// TIA Portal V15.1 export
// export: Created 2024-05-17T05:38:37.8668789Z, ExportSetting WithDefaults, DisplayName Totally Integrated Automation Portal, DisplayVersion V15.1 Update 5, DisplayName TIA Portal Openness, DisplayVersion V15.1 Update 5, DisplayName SINAMICS Startdrive Advanced, DisplayVersion V15.1, DisplayName G130, G150, S120, S150, SINAMICS MV, S210, DisplayVersion V15.1, DisplayName G110M, G120, G120C, G120D, G120P, DisplayVersion V15.1, DisplayName STEP 7 Professional, DisplayVersion V15.1 Update 5, DisplayName STEP 7 Safety, DisplayVersion V15.1, DisplayName WinCC Professional, DisplayVersion V15.1 Update 5, DisplayName SIMATIC Visualization Architect, DisplayVersion V15.1
FUNCTION_BLOCK "LGBMotor2W2S-FC302PN"   // FB6601, FBD
TITLE = LGBMotor2W2S-FC302PN
{ S7_Optimized_Access := 'TRUE' }
AUTHOR : VCC
FAMILY : Actuator
NAME : Danfoss
VERSION : 0.1
// ============================================================================
// This "LMotor2W2S-FC302PN" module is used in applications when a motor 2 way - variable 
// speed equipped with Danfoss FC302 is needed.
// The module contains: a motor loop equipped with 
// "1 Danfoss frequency converter.
// "1 safety switch.
// ============================================================================
// stored: AutoNumber false, IsIECCheckEnabled false, IsRetainMemResEnabled false, MemoryReserve 100, SetENOAutomatically False, UDAEnableTagReadback false
   VAR_INPUT
      I_EnableAlarm { ExternalAccessible := 'False'; ExternalVisible := 'False'; ExternalWritable := 'False'} : Bool;   // Enable alarm
      I_EnablePNReset { ExternalAccessible := 'False'; ExternalVisible := 'False'; ExternalWritable := 'False'} : Bool;   // Enable frequency convertor reset with
      I_AlarmResetPB { ExternalAccessible := 'False'; ExternalVisible := 'False'; ExternalWritable := 'False'} : Bool;   // Alarm reset pushbutton is activated
      I_MotorProtection { ExternalAccessible := 'False'; ExternalVisible := 'False'; ExternalWritable := 'False'} : Bool;   // Motor protection
      I_BrakeProtection { ExternalAccessible := 'False'; ExternalVisible := 'False'; ExternalWritable := 'False'} : Bool;   // Brake protection
      I_SafetySwitch { ExternalAccessible := 'False'; ExternalVisible := 'False'; ExternalWritable := 'False'} : Bool;   // Safety Switch
      I_SafetyOk { ExternalAccessible := 'False'; ExternalVisible := 'False'; ExternalWritable := 'False'} : Bool;   // Safety Ok
      I_MotionStopOk { ExternalAccessible := 'False'; ExternalVisible := 'False'; ExternalWritable := 'False'} : Bool;   // Safety Ok / The motion stop is Ok
      I_Release { ExternalAccessible := 'False'; ExternalVisible := 'False'; ExternalWritable := 'False'} : Bool := TRUE;   // Hold Motor Command
      I_LSpdSetMotorCmd { ExternalAccessible := 'False'; ExternalVisible := 'False'; ExternalWritable := 'False'} : Bool;   // Low speed Set Command from function after interlock
      I_HSpdSetMotorCmd { ExternalAccessible := 'False'; ExternalVisible := 'False'; ExternalWritable := 'False'} : Bool;   // High Speed Set Command from function after Interlock
      I_LSpdResMotorCmd { ExternalAccessible := 'False'; ExternalVisible := 'False'; ExternalWritable := 'False'} : Bool;   // Low speed Reset Command from function after interlock
      I_HSpdResMotorCmd { ExternalAccessible := 'False'; ExternalVisible := 'False'; ExternalWritable := 'False'} : Bool;   // High speed Reset Command from function after Interlock
      I_QuickStop { ExternalAccessible := 'False'; ExternalVisible := 'False'; ExternalWritable := 'False'} : Bool;   // QuickStop function; When FALSE the QuickStop of the Danfoss FC302 is Active
      I_ReleaseBrake { ExternalAccessible := 'False'; ExternalVisible := 'False'; ExternalWritable := 'False'} : Bool;   // Release brake
      I_InitDirection { ExternalAccessible := 'False'; ExternalVisible := 'False'; ExternalWritable := 'False'} : Bool;   // Initialisation of the direction
      I_SetupSelLsb { ExternalAccessible := 'False'; ExternalVisible := 'False'; ExternalWritable := 'False'} : Bool;   // Enable setpoint
      I_SetupSelMsb { ExternalAccessible := 'False'; ExternalVisible := 'False'; ExternalWritable := 'False'} : Bool;   // Enable setpoint
      I_LowSpeed { ExternalAccessible := 'False'; ExternalVisible := 'False'; ExternalWritable := 'False'} : Real;   // Low speed value (set-up %) Reference value for speed, stored in P2000 ot the SINAMICS G120
      I_HighSpeed { ExternalAccessible := 'False'; ExternalVisible := 'False'; ExternalWritable := 'False'} : Real;   // High speed value (set-up %) Reference value for speed, stored in P2000 ot the SINAMICS G120
   END_VAR
   VAR_OUTPUT
      O_BusFault { ExternalAccessible := 'False'; ExternalVisible := 'False'; ExternalWritable := 'False'} : Bool;   // Alarm
      O_MotorProtectionAlarm { ExternalAccessible := 'False'; ExternalVisible := 'False'; ExternalWritable := 'False'} : Bool;   // Motor protection Alarm
      O_BrakeProtectionAlarm { ExternalAccessible := 'False'; ExternalVisible := 'False'; ExternalWritable := 'False'} : Bool;   // Brake protection alarm
      O_SafetySwitchAlarm { ExternalAccessible := 'False'; ExternalVisible := 'False'; ExternalWritable := 'False'} : Bool;   // Safety Switch Alarm
      O_MotionStopWarning { ExternalAccessible := 'False'; ExternalVisible := 'False'; ExternalWritable := 'False'} : Bool;   // Drive fault / Motion Stop warning
      O_Alarm { ExternalAccessible := 'False'; ExternalVisible := 'False'; ExternalWritable := 'False'} : Bool;   // Alarm
      O_Warning { ExternalAccessible := 'False'; ExternalVisible := 'False'; ExternalWritable := 'False'} : Bool;   // Warning
      O_AlarmABCondition { ExternalAccessible := 'False'; ExternalVisible := 'False'; ExternalWritable := 'False'} : Bool;   // Alarm AB condition
      O_Active { ExternalAccessible := 'False'; ExternalVisible := 'False'; ExternalWritable := 'False'} : Bool;   // Motor loop Active
      O_BrakeFunction { ExternalAccessible := 'False'; ExternalVisible := 'False'; ExternalWritable := 'False'} : Bool;   // Brake Function
      O_ReadyForOperation { ExternalAccessible := 'False'; ExternalVisible := 'False'; ExternalWritable := 'False'} : Bool;   // Ready for operation
      O_ActualSpeed { ExternalAccessible := 'False'; ExternalVisible := 'False'; ExternalWritable := 'False'} : Real;   // Actual Speed
   END_VAR
   VAR_IN_OUT
      IO_Modes : "Modes";   // Modes
      H_HMI : "H_HMI";
      "H_GBMotor2W2S-FC302PN" : "H_GBMotor2W2S-FC302PN";
      C_HWSubInput { ExternalAccessible := 'False'; ExternalVisible := 'False'; ExternalWritable := 'False'} : HW_SUBMODULE;   // I/O
      C_HWSubOutput { ExternalAccessible := 'False'; ExternalVisible := 'False'; ExternalWritable := 'False'} : HW_SUBMODULE;   // I/O
      C_EnableCheckSpeed { ExternalAccessible := 'False'; ExternalVisible := 'False'; ExternalWritable := 'False'} : Bool;   // Enable check speed is OK
      C_TimeCheckSpeedOK { ExternalAccessible := 'False'; ExternalVisible := 'False'; ExternalWritable := 'False'} : DInt := 2000;   // Time check speed OK
      C_ReleaseBrakeUsed { ExternalAccessible := 'False'; ExternalVisible := 'False'; ExternalWritable := 'False'} : Bool;   // Release brake used
      C_MotorProtectionUsed { ExternalAccessible := 'False'; ExternalVisible := 'False'; ExternalWritable := 'False'} : Bool;   // Motor Protection used
      C_MotorProtectionNc { ExternalAccessible := 'False'; ExternalVisible := 'False'; ExternalWritable := 'False'} : Bool;   // Motor Protection Normally closed
      C_BrakeProtectionUsed { ExternalAccessible := 'False'; ExternalVisible := 'False'; ExternalWritable := 'False'} : Bool;   // Brake Protection used / Motor Protection used
      C_BrakeProtectionNc { ExternalAccessible := 'False'; ExternalVisible := 'False'; ExternalWritable := 'False'} : Bool;   // Motor Protection Normally closed / Brake Protection Normally closed
      C_SafetySwitchUsed { ExternalAccessible := 'False'; ExternalVisible := 'False'; ExternalWritable := 'False'} : Bool;   // Safety switch used
      C_SafetySwitchNc { ExternalAccessible := 'False'; ExternalVisible := 'False'; ExternalWritable := 'False'} : Bool;   // Safety switch Normally closed
      C_MotionStopUsed { ExternalAccessible := 'False'; ExternalVisible := 'False'; ExternalWritable := 'False'} : Bool;   // Motion Stop used
   END_VAR
   VAR
      Start { ExternalAccessible := 'False'; ExternalVisible := 'False'; ExternalWritable := 'False'} : Bool;   // Start
      Reverse { ExternalAccessible := 'False'; ExternalVisible := 'False'; ExternalWritable := 'False'} : Bool;   // Reverse
      MotorProtectionAlarm { ExternalAccessible := 'False'; ExternalVisible := 'False'; ExternalWritable := 'False'} : Bool;   // Motor protection Alarm
      BrakeProtectionAlarm { ExternalAccessible := 'False'; ExternalVisible := 'False'; ExternalWritable := 'False'} : Bool;   // Brake protection alarm
      CheckSpeedOK { ExternalAccessible := 'False'; ExternalVisible := 'False'; ExternalWritable := 'False'} : Bool;   // After this time the speed has to be reached
      SafetySwitchAlarm { ExternalAccessible := 'False'; ExternalVisible := 'False'; ExternalWritable := 'False'} : Bool;   // Safety Switch Alarm
      MotorProtectionAlarmABCond { ExternalAccessible := 'False'; ExternalVisible := 'False'; ExternalWritable := 'False'} : Bool;   // Motor protection Alarm condition
      BrakeProtectionAlarmABCond { ExternalAccessible := 'False'; ExternalVisible := 'False'; ExternalWritable := 'False'} : Bool;   // Brake protection alarm condition
      SafetySwitchAlarmABCond { ExternalAccessible := 'False'; ExternalVisible := 'False'; ExternalWritable := 'False'} : Bool;   // Safety Switch Alarm condition
      FC302PNAlarm { ExternalAccessible := 'False'; ExternalVisible := 'False'; ExternalWritable := 'False'} : Bool;
      FC302PNAlarmABCond { ExternalAccessible := 'False'; ExternalVisible := 'False'; ExternalWritable := 'False'} : Bool;
      MotionStopWarning { ExternalAccessible := 'False'; ExternalVisible := 'False'; ExternalWritable := 'False'} : Bool;   // Drive fault alarm / Motion Stop warning
      Active { ExternalAccessible := 'False'; ExternalVisible := 'False'; ExternalWritable := 'False'} : Bool;
      SpeedSetPoint { ExternalAccessible := 'False'; ExternalVisible := 'False'; ExternalWritable := 'False'} : Real;
      ControlReady { ExternalAccessible := 'False'; ExternalVisible := 'False'; ExternalWritable := 'False'} : Bool;
      DriveReady { ExternalAccessible := 'False'; ExternalVisible := 'False'; ExternalWritable := 'False'} : Bool;
      CoastingReady { ExternalAccessible := 'False'; ExternalVisible := 'False'; ExternalWritable := 'False'} : Bool;
      Trip { ExternalAccessible := 'False'; ExternalVisible := 'False'; ExternalWritable := 'False'} : Bool;
      Error { ExternalAccessible := 'False'; ExternalVisible := 'False'; ExternalWritable := 'False'} : Bool;
      TripLock { ExternalAccessible := 'False'; ExternalVisible := 'False'; ExternalWritable := 'False'} : Bool;
      Warning { ExternalAccessible := 'False'; ExternalVisible := 'False'; ExternalWritable := 'False'} : Bool;
      SpeedOK { ExternalAccessible := 'False'; ExternalVisible := 'False'; ExternalWritable := 'False'} : Bool;
      BusControl { ExternalAccessible := 'False'; ExternalVisible := 'False'; ExternalWritable := 'False'} : Bool;
      FrequencyLimit { ExternalAccessible := 'False'; ExternalVisible := 'False'; ExternalWritable := 'False'} : Bool;
      InOperation { ExternalAccessible := 'False'; ExternalVisible := 'False'; ExternalWritable := 'False'} : Bool;
      Autostart { ExternalAccessible := 'False'; ExternalVisible := 'False'; ExternalWritable := 'False'} : Bool;
      VoltageLimitExceed { ExternalAccessible := 'False'; ExternalVisible := 'False'; ExternalWritable := 'False'} : Bool;
      TorqueLimitExceed { ExternalAccessible := 'False'; ExternalVisible := 'False'; ExternalWritable := 'False'} : Bool;
      TimerLimitExceed { ExternalAccessible := 'False'; ExternalVisible := 'False'; ExternalWritable := 'False'} : Bool;
      ActualSpeed { ExternalAccessible := 'False'; ExternalVisible := 'False'; ExternalWritable := 'False'} : Real;
      _MotorProtection { ExternalAccessible := 'False'; ExternalVisible := 'False'; ExternalWritable := 'False'} : "L1AlarmMultiIn";   // FB
      _BrakeProtection { ExternalAccessible := 'False'; ExternalVisible := 'False'; ExternalWritable := 'False'} : "L1AlarmMultiIn";   // FB
      _SafetySwitch { ExternalAccessible := 'False'; ExternalVisible := 'False'; ExternalWritable := 'False'} : "L1AlarmMultiIn";   // FB
      _FC302PNAlarm { ExternalAccessible := 'False'; ExternalVisible := 'False'; ExternalWritable := 'False'} : "L1AlarmMultiIn";   // FB
      _FC302PN { ExternalAccessible := 'False'; ExternalVisible := 'False'; ExternalWritable := 'False'} : "LGBDanfoss-FC302PN";   // FB
      _MotionStop { ExternalAccessible := 'False'; ExternalVisible := 'False'; ExternalWritable := 'False'} : "L1AlarmMultiIn";   // FB
      _SpeedOKTimer { ExternalAccessible := 'False'; ExternalVisible := 'False'; ExternalWritable := 'False'} : "LTimer";   // Timer
   END_VAR
   VAR_TEMP   // added for the SCL form of the ladder/FBD networks
      _w1 : Bool;
   END_VAR
BEGIN

REGION Network 1: **** 2.2 - Alarms - Alarms Generation **** Motor Safety switch Alarm
   // Motor Safety switch Alarm
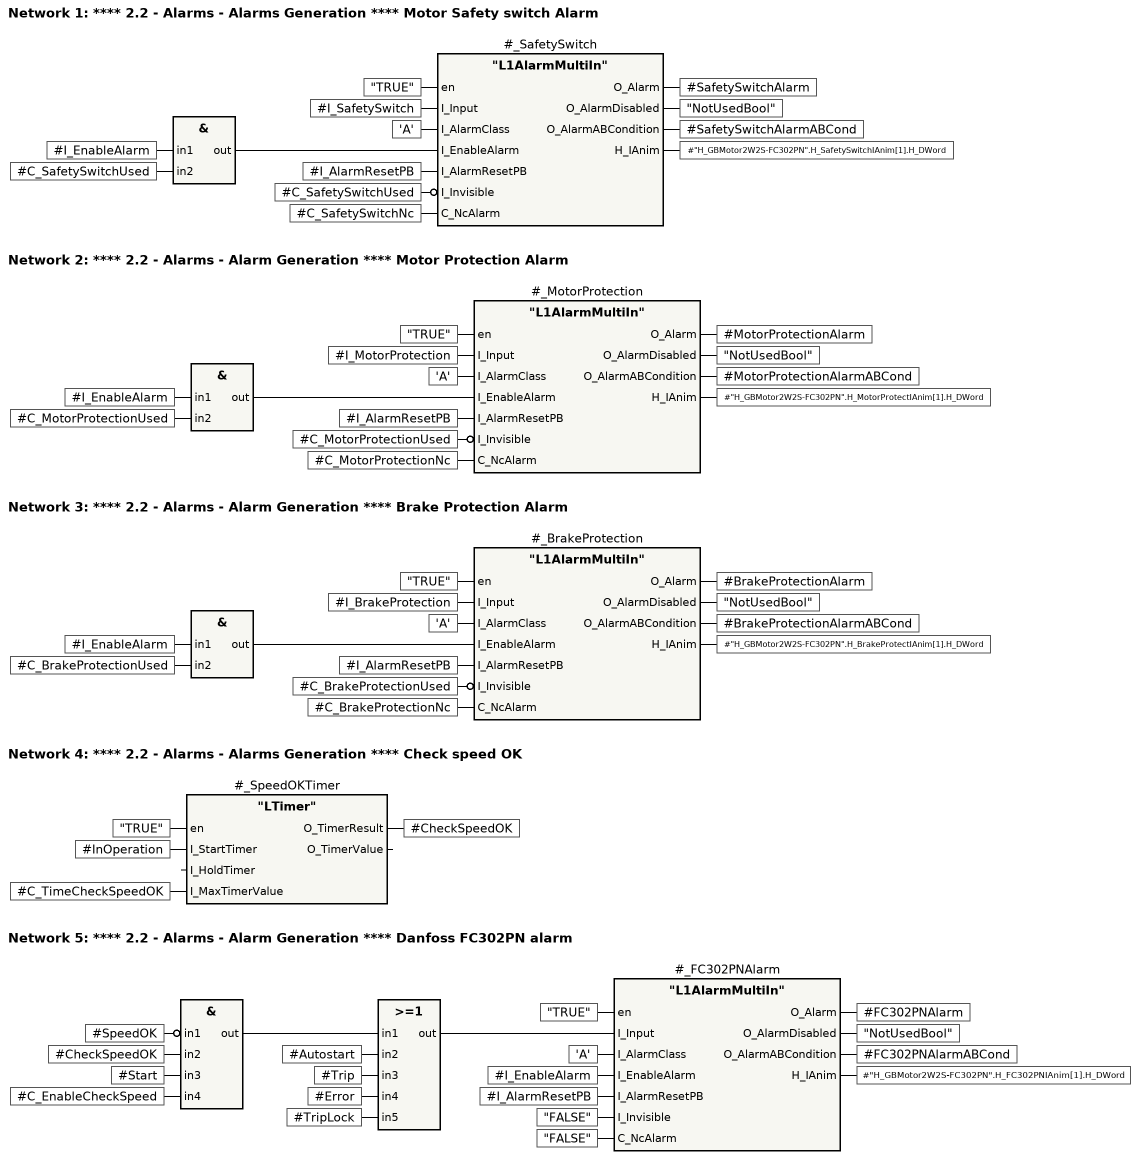
   IF "TRUE" THEN
       #_SafetySwitch(I_Input := #I_SafetySwitch,   // "L1AlarmMultiIn"
                      I_AlarmClass := 'A',
                      I_EnableAlarm := #I_EnableAlarm AND #C_SafetySwitchUsed,
                      I_AlarmResetPB := #I_AlarmResetPB,
                      I_Invisible := NOT #C_SafetySwitchUsed,
                      C_NcAlarm := #C_SafetySwitchNc,
                      O_Alarm => #SafetySwitchAlarm,
                      O_AlarmDisabled => "NotUsedBool",
                      O_AlarmABCondition => #SafetySwitchAlarmABCond,
                      H_IAnim => #"H_GBMotor2W2S-FC302PN".H_SafetySwitchIAnim[1].H_DWord);
   END_IF;
END_REGION

REGION Network 2: **** 2.2 - Alarms - Alarm Generation **** Motor Protection Alarm
   // Motor Protection Alarm
   IF "TRUE" THEN
       #_MotorProtection(I_Input := #I_MotorProtection,   // "L1AlarmMultiIn"
                         I_AlarmClass := 'A',
                         I_EnableAlarm := #I_EnableAlarm AND #C_MotorProtectionUsed,
                         I_AlarmResetPB := #I_AlarmResetPB,
                         I_Invisible := NOT #C_MotorProtectionUsed,
                         C_NcAlarm := #C_MotorProtectionNc,
                         O_Alarm => #MotorProtectionAlarm,
                         O_AlarmDisabled => "NotUsedBool",
                         O_AlarmABCondition => #MotorProtectionAlarmABCond,
                         H_IAnim => #"H_GBMotor2W2S-FC302PN".H_MotorProtectIAnim[1].H_DWord);
   END_IF;
END_REGION

REGION Network 3: **** 2.2 - Alarms - Alarm Generation **** Brake Protection Alarm
   // Brake Protection Alarm
   IF "TRUE" THEN
       #_BrakeProtection(I_Input := #I_BrakeProtection,   // "L1AlarmMultiIn"
                         I_AlarmClass := 'A',
                         I_EnableAlarm := #I_EnableAlarm AND #C_BrakeProtectionUsed,
                         I_AlarmResetPB := #I_AlarmResetPB,
                         I_Invisible := NOT #C_BrakeProtectionUsed,
                         C_NcAlarm := #C_BrakeProtectionNc,
                         O_Alarm => #BrakeProtectionAlarm,
                         O_AlarmDisabled => "NotUsedBool",
                         O_AlarmABCondition => #BrakeProtectionAlarmABCond,
                         H_IAnim => #"H_GBMotor2W2S-FC302PN".H_BrakeProtectIAnim[1].H_DWord);
   END_IF;
END_REGION

REGION Network 4: **** 2.2 - Alarms - Alarms Generation **** Check speed OK
   // Timer check speed is OK
   IF "TRUE" THEN
       #_SpeedOKTimer(I_StartTimer := #InOperation,   // "LTimer"
                      I_MaxTimerValue := #C_TimeCheckSpeedOK,
                      O_TimerResult => #CheckSpeedOK);
   END_IF;
END_REGION

REGION Network 5: **** 2.2 - Alarms - Alarm Generation **** Danfoss FC302PN alarm
   // Danfoss FC302PN alarm
   IF "TRUE" THEN
       #_FC302PNAlarm(I_Input := (NOT #SpeedOK AND #CheckSpeedOK AND #Start AND #C_EnableCheckSpeed) OR #Autostart OR #Trip OR #Error OR #TripLock,   // "L1AlarmMultiIn"
                      I_AlarmClass := 'A',
                      I_EnableAlarm := #I_EnableAlarm,
                      I_AlarmResetPB := #I_AlarmResetPB,
                      I_Invisible := "FALSE",
                      C_NcAlarm := "FALSE",
                      O_Alarm => #FC302PNAlarm,
                      O_AlarmDisabled => "NotUsedBool",
                      O_AlarmABCondition => #FC302PNAlarmABCond,
                      H_IAnim => #"H_GBMotor2W2S-FC302PN".H_FC302PNIAnim[1].H_DWord);
   END_IF;
END_REGION

REGION Network 6: **** 2.2 - Alarms - Alarm Generation **** MotionStop Warning
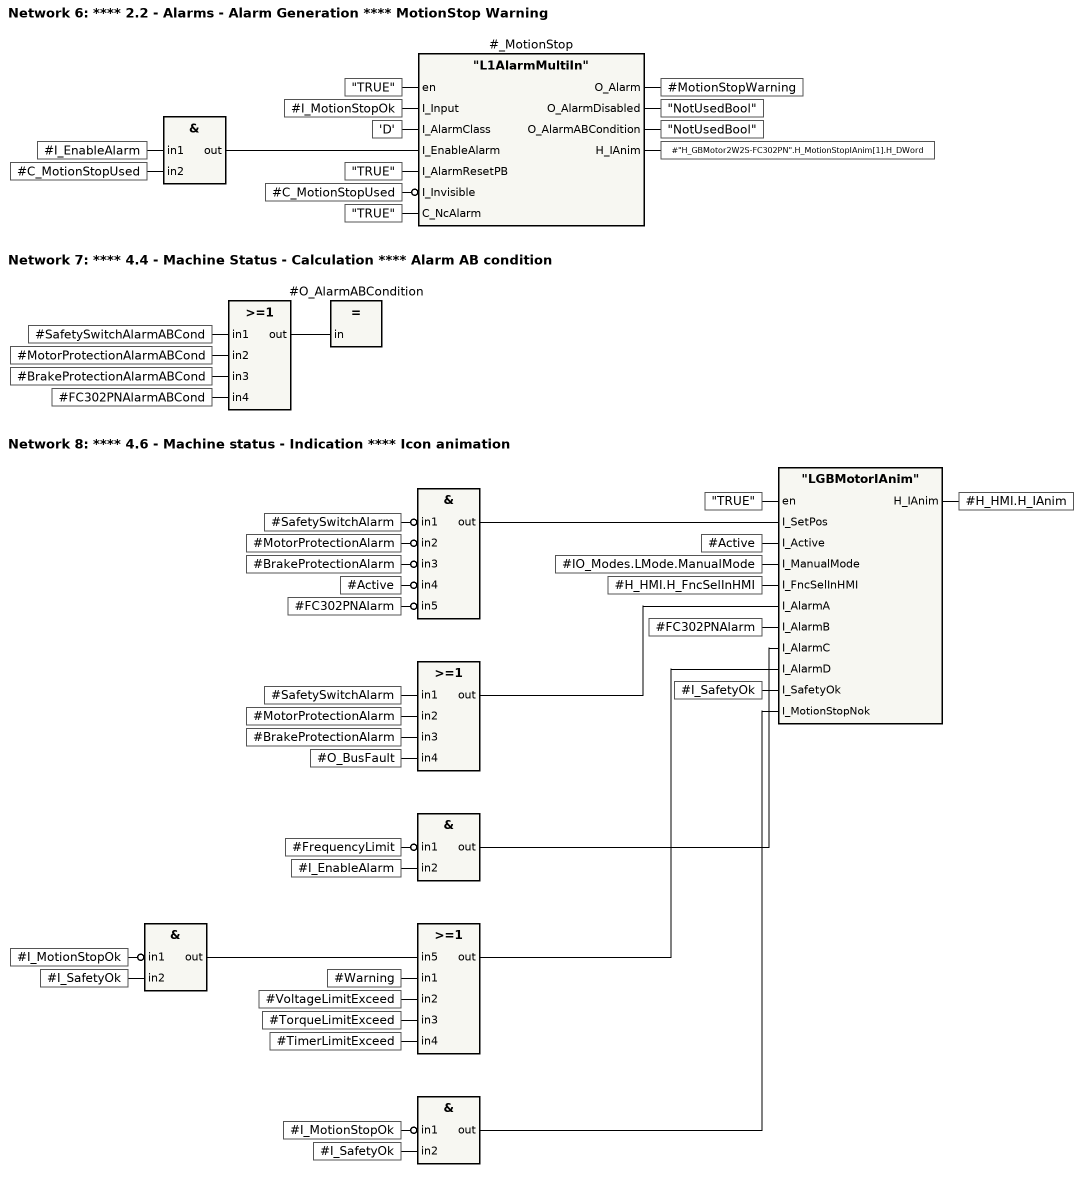
   IF "TRUE" THEN
       #_MotionStop(I_Input := #I_MotionStopOk,   // "L1AlarmMultiIn"
                    I_AlarmClass := 'D',
                    I_EnableAlarm := #I_EnableAlarm AND #C_MotionStopUsed,
                    I_AlarmResetPB := "TRUE",
                    I_Invisible := NOT #C_MotionStopUsed,
                    C_NcAlarm := "TRUE",
                    O_Alarm => #MotionStopWarning,
                    O_AlarmDisabled => "NotUsedBool",
                    O_AlarmABCondition => "NotUsedBool",
                    H_IAnim => #"H_GBMotor2W2S-FC302PN".H_MotionStopIAnim[1].H_DWord);
   END_IF;
END_REGION

REGION Network 7: **** 4.4 - Machine Status - Calculation **** Alarm AB condition
   // Alarm AB condition
   #O_AlarmABCondition := #SafetySwitchAlarmABCond OR #MotorProtectionAlarmABCond OR #BrakeProtectionAlarmABCond OR #FC302PNAlarmABCond;
END_REGION

REGION Network 8: **** 4.6 - Machine status - Indication **** Icon animation
   // Icon animation
   IF "TRUE" THEN
       "LGBMotorIAnim"(I_SetPos := NOT #SafetySwitchAlarm AND NOT #MotorProtectionAlarm AND NOT #BrakeProtectionAlarm AND NOT #Active AND NOT #FC302PNAlarm,
                       I_Active := #Active,
                       I_ManualMode := #IO_Modes.LMode.ManualMode,
                       I_FncSelInHMI := #H_HMI.H_FncSelInHMI,
                       I_AlarmA := #SafetySwitchAlarm OR #MotorProtectionAlarm OR #BrakeProtectionAlarm OR #O_BusFault,
                       I_AlarmB := #FC302PNAlarm,
                       I_AlarmC := NOT #FrequencyLimit AND #I_EnableAlarm,
                       I_AlarmD := (NOT #I_MotionStopOk AND #I_SafetyOk) OR #Warning OR #VoltageLimitExceed OR #TorqueLimitExceed OR #TimerLimitExceed,
                       I_SafetyOk := #I_SafetyOk,
                       I_MotionStopNok := NOT #I_MotionStopOk AND #I_SafetyOk,
                       H_IAnim => #H_HMI.H_IAnim);
   END_IF;
END_REGION

REGION Network 9: **** 4.6 - Machine status - Indication **** Animation
   // Animation
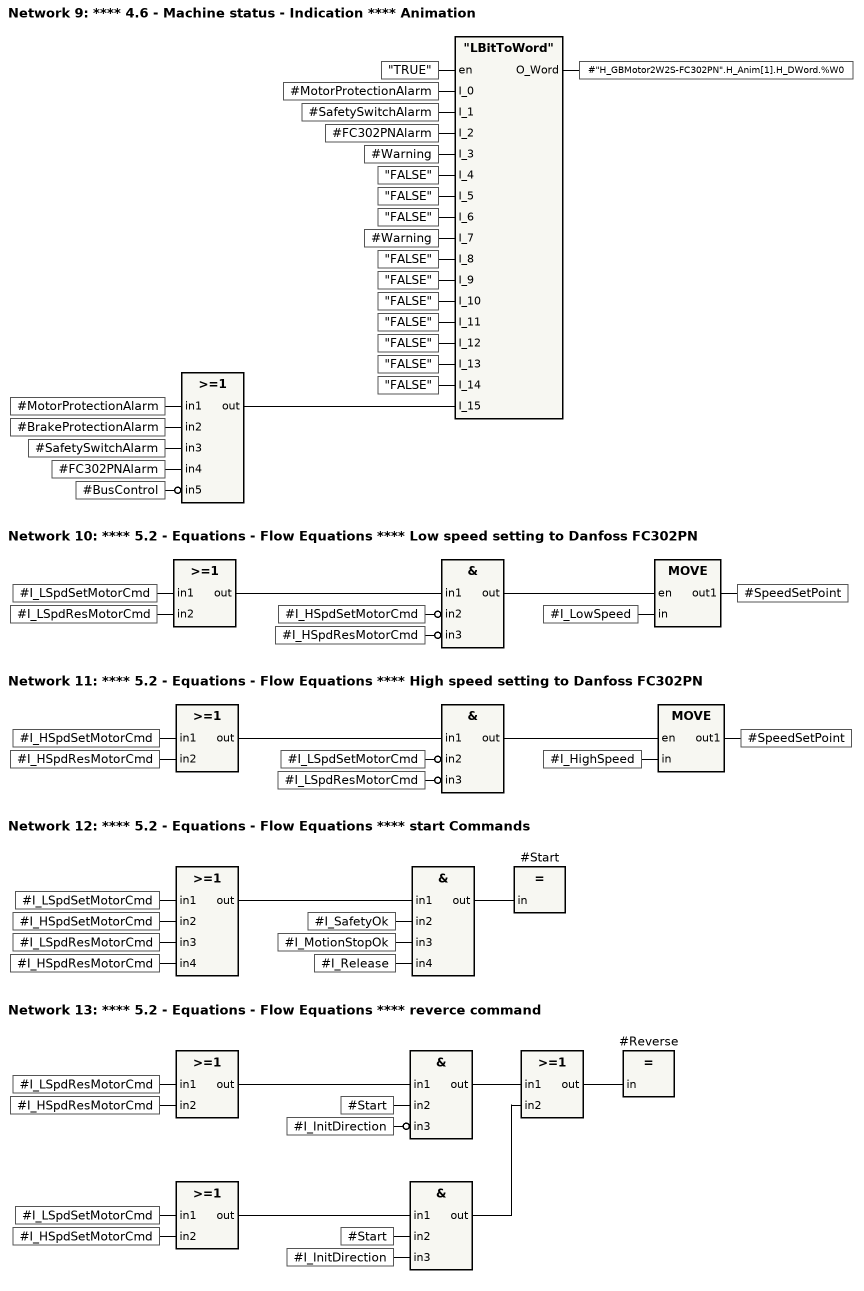
   IF "TRUE" THEN
       "LBitToWord"(I_0 := #MotorProtectionAlarm,
                    I_1 := #SafetySwitchAlarm,
                    I_2 := #FC302PNAlarm,
                    I_3 := #Warning,
                    I_4 := "FALSE",
                    I_5 := "FALSE",
                    I_6 := "FALSE",
                    I_7 := #Warning,
                    I_8 := "FALSE",
                    I_9 := "FALSE",
                    I_10 := "FALSE",
                    I_11 := "FALSE",
                    I_12 := "FALSE",
                    I_13 := "FALSE",
                    I_14 := "FALSE",
                    I_15 := #MotorProtectionAlarm OR #BrakeProtectionAlarm OR #SafetySwitchAlarm OR #FC302PNAlarm OR NOT #BusControl,
                    O_Word => #"H_GBMotor2W2S-FC302PN".H_Anim[1].H_DWord.%W0);
   END_IF;
END_REGION

REGION Network 10: **** 5.2 - Equations - Flow Equations **** Low speed setting to Danfoss FC302PN
   // Low speed setting to Danfoss
   IF (#I_LSpdSetMotorCmd OR #I_LSpdResMotorCmd) AND NOT #I_HSpdSetMotorCmd AND NOT #I_HSpdResMotorCmd THEN
       #SpeedSetPoint := #I_LowSpeed;
   END_IF;
END_REGION

REGION Network 11: **** 5.2 - Equations - Flow Equations **** High speed setting to Danfoss FC302PN
   // High speed setting to Danfoss
   IF (#I_HSpdSetMotorCmd OR #I_HSpdResMotorCmd) AND NOT #I_LSpdSetMotorCmd AND NOT #I_LSpdResMotorCmd THEN
       #SpeedSetPoint := #I_HighSpeed;
   END_IF;
END_REGION

REGION Network 12: **** 5.2 - Equations - Flow Equations **** start Commands
   // Send Drive start Commands
   #Start := (#I_LSpdSetMotorCmd OR #I_HSpdSetMotorCmd OR #I_LSpdResMotorCmd OR #I_HSpdResMotorCmd) AND #I_SafetyOk AND #I_MotionStopOk AND #I_Release;
END_REGION

REGION Network 13: **** 5.2 - Equations - Flow Equations **** reverce command
   // Send drive reverce command
   #Reverse := ((#I_LSpdResMotorCmd OR #I_HSpdResMotorCmd) AND #Start AND NOT #I_InitDirection) OR ((#I_LSpdSetMotorCmd OR #I_HSpdSetMotorCmd) AND #Start AND #I_InitDirection);
END_REGION

REGION Network 14: **** 5.2 - Equations - Flow Equations **** Active
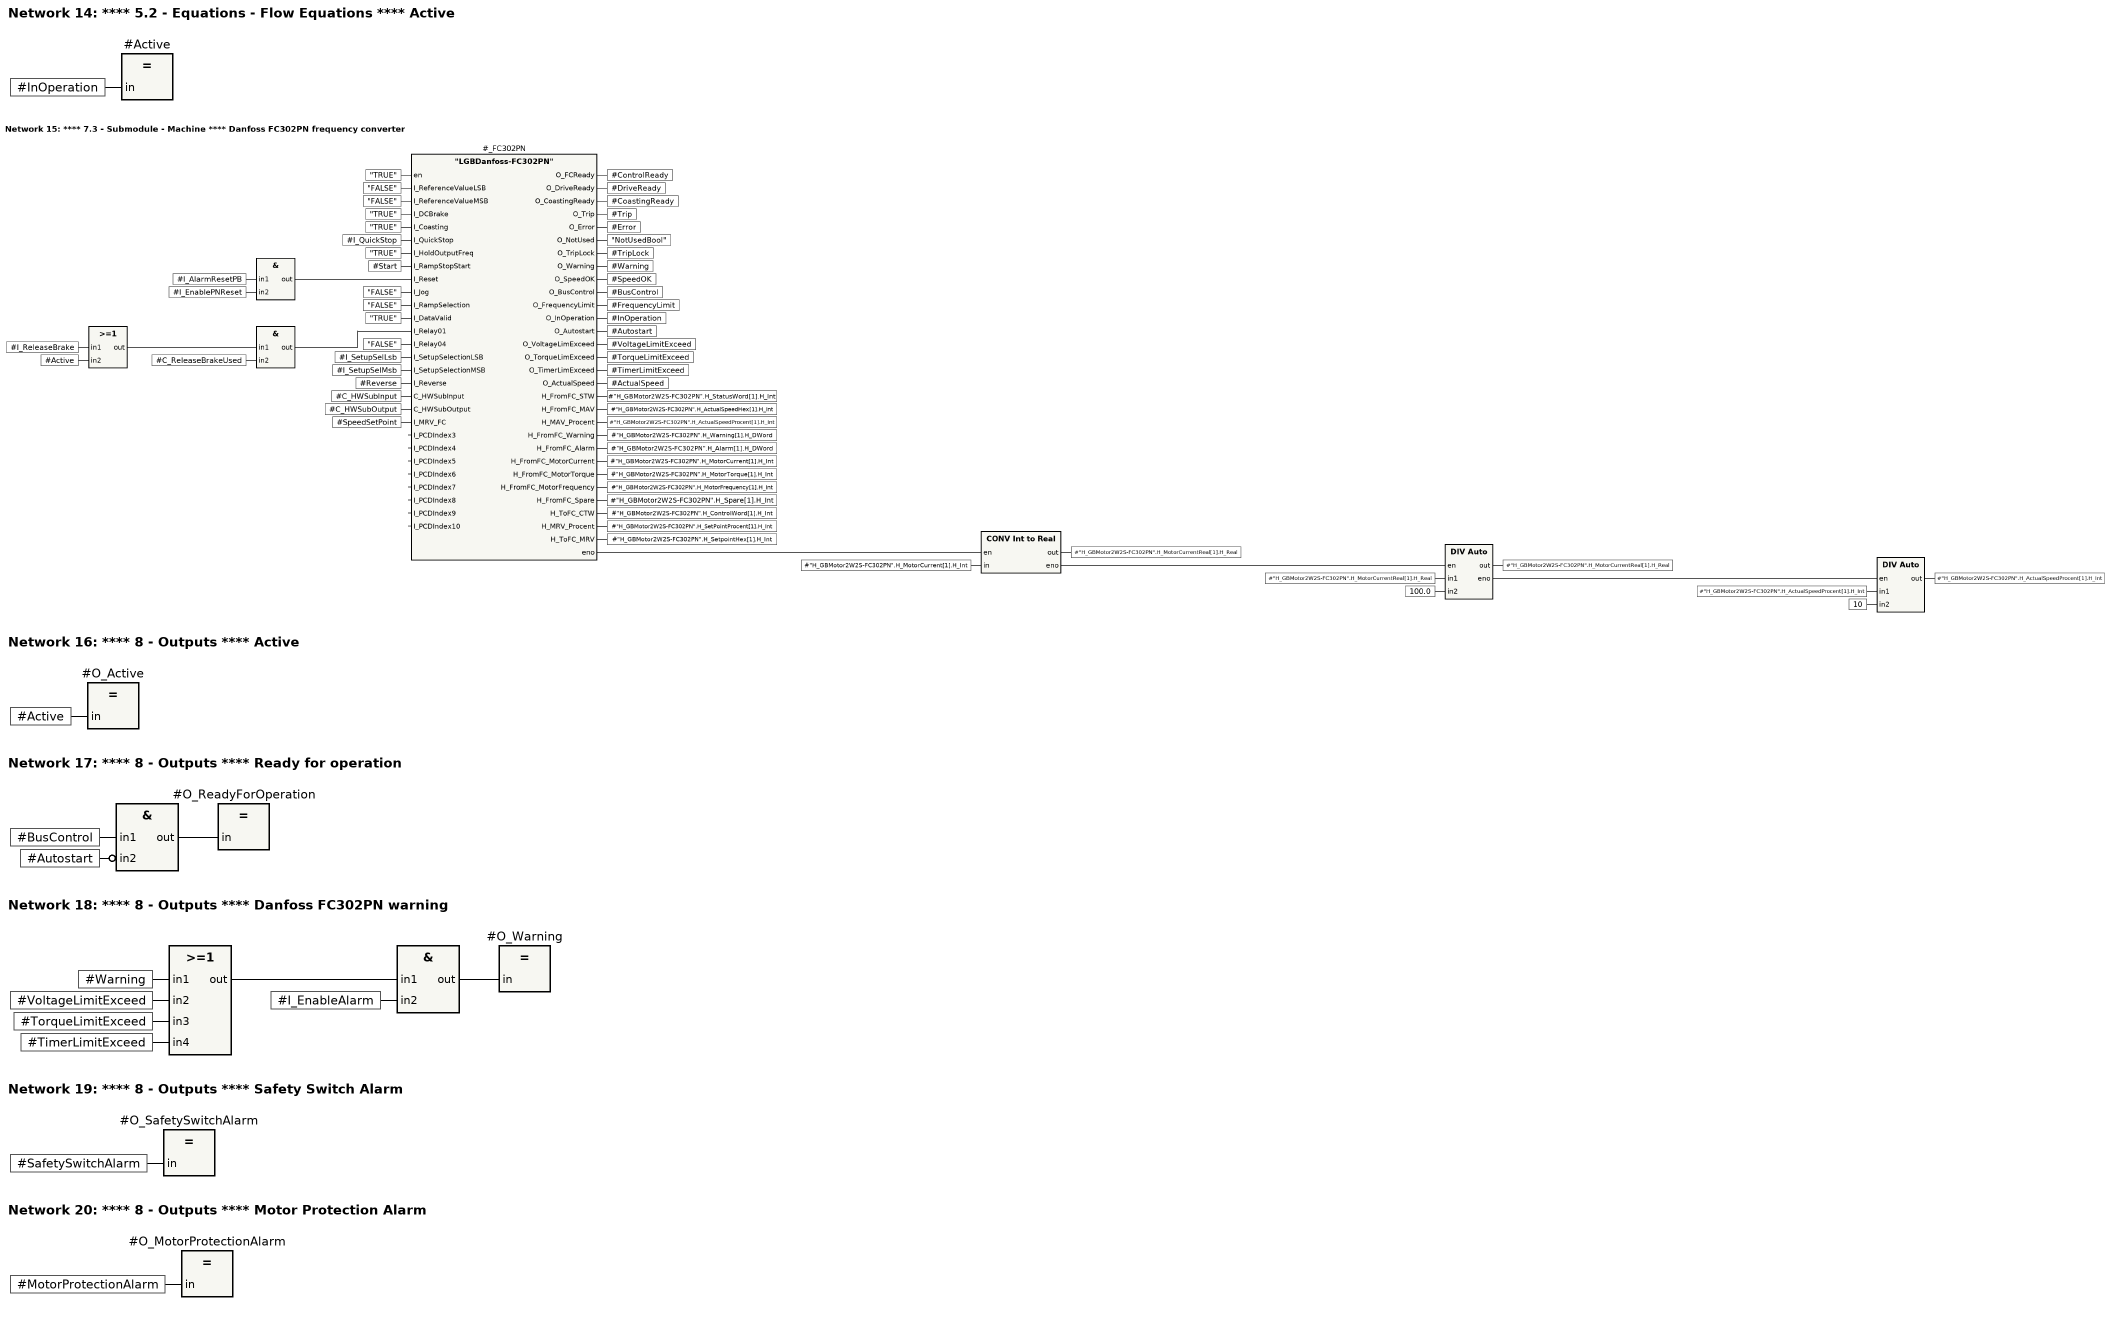
   #Active := #InOperation;
END_REGION

REGION Network 15: **** 7.3 - Submodule - Machine **** Danfoss FC302PN frequency converter
   // Frequency controller
   #_FC302PN(EN := "TRUE",   // "LGBDanfoss-FC302PN"
             I_ReferenceValueLSB := "FALSE",
             I_ReferenceValueMSB := "FALSE",
             I_DCBrake := "TRUE",
             I_Coasting := "TRUE",
             I_QuickStop := #I_QuickStop,
             I_HoldOutputFreq := "TRUE",
             I_RampStopStart := #Start,
             I_Reset := #I_AlarmResetPB AND #I_EnablePNReset,
             I_Jog := "FALSE",
             I_RampSelection := "FALSE",
             I_DataValid := "TRUE",
             I_Relay01 := (#I_ReleaseBrake OR #Active) AND #C_ReleaseBrakeUsed,
             I_Relay04 := "FALSE",
             I_SetupSelectionLSB := #I_SetupSelLsb,
             I_SetupSelectionMSB := #I_SetupSelMsb,
             I_Reverse := #Reverse,
             C_HWSubInput := #C_HWSubInput,
             C_HWSubOutput := #C_HWSubOutput,
             I_MRV_FC := #SpeedSetPoint,
             O_FCReady => #ControlReady,
             O_DriveReady => #DriveReady,
             O_CoastingReady => #CoastingReady,
             O_Trip => #Trip,
             O_Error => #Error,
             O_NotUsed => "NotUsedBool",
             O_TripLock => #TripLock,
             O_Warning => #Warning,
             O_SpeedOK => #SpeedOK,
             O_BusControl => #BusControl,
             O_FrequencyLimit => #FrequencyLimit,
             O_InOperation => #InOperation,
             O_Autostart => #Autostart,
             O_VoltageLimExceed => #VoltageLimitExceed,
             O_TorqueLimExceed => #TorqueLimitExceed,
             O_TimerLimExceed => #TimerLimitExceed,
             O_ActualSpeed => #ActualSpeed,
             H_FromFC_STW => #"H_GBMotor2W2S-FC302PN".H_StatusWord[1].H_Int,
             H_FromFC_MAV => #"H_GBMotor2W2S-FC302PN".H_ActualSpeedHex[1].H_Int,
             H_MAV_Procent => #"H_GBMotor2W2S-FC302PN".H_ActualSpeedProcent[1].H_Int,
             H_FromFC_Warning => #"H_GBMotor2W2S-FC302PN".H_Warning[1].H_DWord,
             H_FromFC_Alarm => #"H_GBMotor2W2S-FC302PN".H_Alarm[1].H_DWord,
             H_FromFC_MotorCurrent => #"H_GBMotor2W2S-FC302PN".H_MotorCurrent[1].H_Int,
             H_FromFC_MotorTorque => #"H_GBMotor2W2S-FC302PN".H_MotorTorque[1].H_Int,
             H_FromFC_MotorFrequency => #"H_GBMotor2W2S-FC302PN".H_MotorFrequency[1].H_Int,
             H_FromFC_Spare => #"H_GBMotor2W2S-FC302PN".H_Spare[1].H_Int,
             H_ToFC_CTW => #"H_GBMotor2W2S-FC302PN".H_ControlWord[1].H_Int,
             H_MRV_Procent => #"H_GBMotor2W2S-FC302PN".H_SetPointProcent[1].H_Int,
             H_ToFC_MRV => #"H_GBMotor2W2S-FC302PN".H_SetpointHex[1].H_Int,
             ENO => #_w1);
   IF #_w1 THEN
       #"H_GBMotor2W2S-FC302PN".H_MotorCurrentReal[1].H_Real := INT_TO_REAL(#"H_GBMotor2W2S-FC302PN".H_MotorCurrent[1].H_Int);
       #"H_GBMotor2W2S-FC302PN".H_MotorCurrentReal[1].H_Real := #"H_GBMotor2W2S-FC302PN".H_MotorCurrentReal[1].H_Real / 100.0;
       #"H_GBMotor2W2S-FC302PN".H_ActualSpeedProcent[1].H_Int := #"H_GBMotor2W2S-FC302PN".H_ActualSpeedProcent[1].H_Int / 10;
   END_IF;
END_REGION

REGION Network 16: **** 8 - Outputs **** Active
   // Active
   #O_Active := #Active;
END_REGION

REGION Network 17: **** 8 - Outputs **** Ready for operation
   // Ready for operation
   #O_ReadyForOperation := #BusControl AND NOT #Autostart;
END_REGION

REGION Network 18: **** 8 - Outputs **** Danfoss FC302PN warning
   // Danfoss FC302PN warning
   #O_Warning := (#Warning OR #VoltageLimitExceed OR #TorqueLimitExceed OR #TimerLimitExceed) AND #I_EnableAlarm;
END_REGION

REGION Network 19: **** 8 - Outputs **** Safety Switch Alarm
   // Safety Switch Alarm
   #O_SafetySwitchAlarm := #SafetySwitchAlarm;
END_REGION

REGION Network 20: **** 8 - Outputs **** Motor Protection Alarm
   // Motor protection Alarm
   #O_MotorProtectionAlarm := #MotorProtectionAlarm;
END_REGION

REGION Network 21: **** 8 - Outputs **** Motor Protection Alarm / **** 8 - Outputs **** Brake Protection Alarm
   // Motor Protection Alarm / Brake Protection Alarm
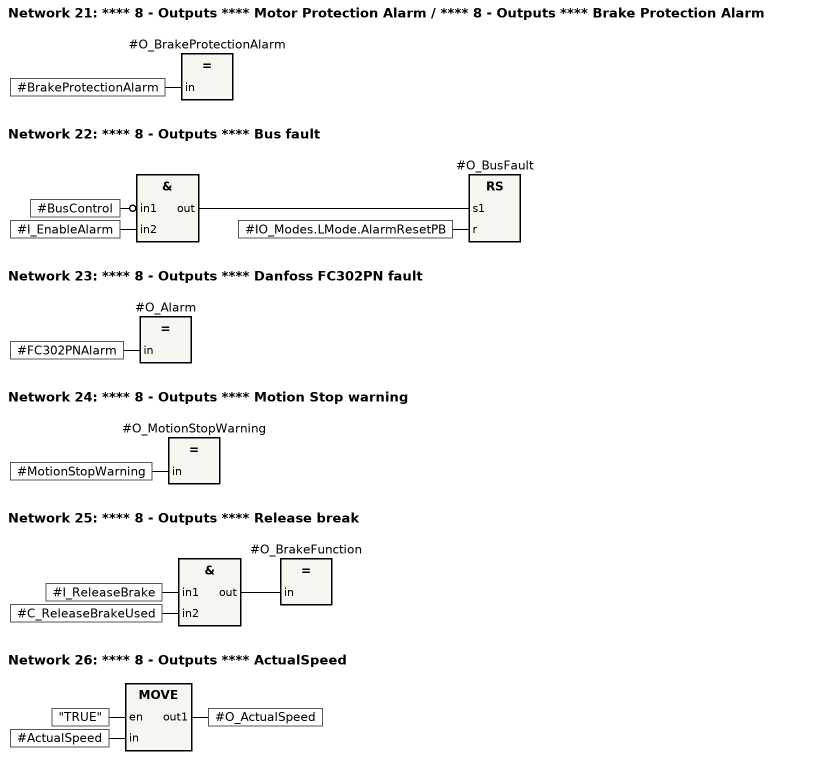
   #O_BrakeProtectionAlarm := #BrakeProtectionAlarm;
END_REGION

REGION Network 22: **** 8 - Outputs **** Bus fault
   // Danfoss fault
   IF #IO_Modes.LMode.AlarmResetPB THEN
       #O_BusFault := FALSE;   // RS flip-flop
   END_IF;
   IF NOT #BusControl AND #I_EnableAlarm THEN #O_BusFault := TRUE; END_IF;
END_REGION

REGION Network 23: **** 8 - Outputs **** Danfoss FC302PN fault
   // Danfoss fault
   #O_Alarm := #FC302PNAlarm;
END_REGION

REGION Network 24: **** 8 - Outputs **** Motion Stop warning
   #O_MotionStopWarning := #MotionStopWarning;
END_REGION

REGION Network 25: **** 8 - Outputs **** Release break
   // Release break of frequency controller (Option)
   #O_BrakeFunction := #I_ReleaseBrake AND #C_ReleaseBrakeUsed;
END_REGION

REGION Network 26: **** 8 - Outputs **** ActualSpeed
   // ActualSpeed
   IF "TRUE" THEN #O_ActualSpeed := #ActualSpeed; END_IF;
END_REGION
END_FUNCTION_BLOCK
